FUNCTION F_TimeAsString : T_MaxString
VAR_INPUT
    TimeStruct : TIMESTRUCT;
END_VAR

F_TimeAsString := F_FormatString3(
                      Format := '%.2d:%.2d:%.2d',
                      arg1   := F_WORD(TimeStruct.wHour),
                      arg2   := F_WORD(TimeStruct.wMinute),
                      arg3   := F_WORD(TimeStruct.wSecond));

END_FUNCTION

(* stored: Version 1.1.0.1, ProductVersion 3.1.4024.3
   POU F_TimeAsString: Id {7575e187-8a5c-007c-25dd-194c79fd74e7}, SpecialFunc None *)
